// TwinCAT 3 PLC project Test
// ProgramVersion: 3.1.4020.10
// libraries:
//   Tc2_MC2, * (Beckhoff Automation GmbH)
//   Tc2_SerialCom, * (Beckhoff Automation GmbH)
//   Tc2_Standard, * (Beckhoff Automation GmbH)
//   Tc2_System, * (Beckhoff Automation GmbH)
//   Tc2_TcpIp, * (Beckhoff Automation GmbH)
//   Tc2_Utilities, * (Beckhoff Automation GmbH)
//   Tc3_Module, * (Beckhoff Automation GmbH)
// project tree:
//   DUTs/ ASCII.TcDUT, Boat.TcDUT
//   GVLs/ GVL_Const.TcGVL, IO.TcGVL
//   / PlcTask.TcTTO
//   POUs/ MAIN.TcPOU
//   POUs/model/ FB_AXIS.TcPOU, FB_Object.TcPOU, FB_RobotCom.TcPOU, FB_String.TcPOU, F_Messages.TcPOU, FB_TP.TcPOU, PRG_Com.TcPOU

CONFIGURATION Test
    RESOURCE PLC ON TwinCAT3
        TASK PlcTask(INTERVAL := T#10ms, PRIORITY := 20);
        PROGRAM MAIN WITH PlcTask : MAIN;
    END_RESOURCE
END_CONFIGURATION

// ---- DUTs/ASCII.TcDUT
TYPE ASCII :
STRUCT	
	AscByte			:ARRAY[1..5] OF BYTE;
END_STRUCT
END_TYPE

// ---- DUTs/Boat.TcDUT
//{attribute 'pack_mode' :='1'}
TYPE Boat :
STRUCT
	ID				: LREAL;			//ID
	CoolTime		: LREAL ;			//冷却时间
	BoatErrHandle	: LREAL ;			//报警舟处理：0未确认1回炉工艺2到自动化检查
	UseTimes		: LREAL ;			//使用次数
	bWaferLoad		: BOOL ;			//装片
	bJobDone		: BOOL ;			//工艺完成
	bCool			: BOOL ;			//冷却完成
	bNeedWash		: BOOL ;			//清洗		
	bError			: BOOL ;			//报警
	bReserve		: BOOL ;			//新舟 	
END_STRUCT
END_TYPE

// ---- GVLs/GVL_Const.TcGVL
{attribute 'qualified_only'}
VAR_GLOBAL
	
END_VAR

// ---- GVLs/IO.TcGVL
{attribute 'qualified_only'}
VAR_GLOBAL
	//Axisx_io: Tc2_MC2.AXIS_REF;
	IoTest 		AT %IB100 		: ARRAY[1..20] OF UINT;
	IoTest1		AT %QB100 	: ARRAY[1..20] OF UINT;
END_VAR

// ---- POUs/MAIN.TcPOU
PROGRAM MAIN
VAR
	AxisX				:FB_AXIS;
	Jogtest				:BOOL;
	bJOGPlus			:BOOL;
	bpower				:BOOL;
	ss,ss1				:STRING;
	var1,var2,var3		:INT;
	rvar1				:LREAL;
	iloop				:INT;
	rlayer				:REAL;
	bpttest				:BOOL;
	pttest1				:FB_TP;
	ptTest				:TP;
	ptout				:BOOL;
	ptin				:BOOL;
	rpttest				:R_TRIG;
	ttest				:TIME;
	bGetNetId			:BOOL:=FALSE;
	NullId				: T_AmsNetID:='0.0.0.0.0.0';
	bEnableCerDis		: BOOL;
	NT_StartProcess		: NT_StartProcess;
	NetId: T_AmsNetID;
	GetLocalAmsNetId: FB_GetLocalAmsNetId;	
	CPJ_DataTrans		:FB_RobotCom;
	PlcTaskSysInfo		: PlcTaskSystemInfo ;			//系统任务信息	
	ss11:STRING(6);
	ss12:STRING(1);
	Out_BoatID:BYTE;
	W:WORD;
	mystr:FB_String;
	i:UINT;
	StrToSend:STRING;
	I1:INT;
END_VAR

//W:=10;
//ss:=WORD_TO_HEXSTR(in:= W, iPrecision:= 2, bLoCase:= FALSE);
//M_PT();
//Init();
//M_Axis();
//CPJ_DataTrans.M_Run();
//mystr.A_Run();
//StrToSend:= CONCAT(CONCAT(CONCAT(CONCAT('@0',INT_TO_STRING(I1)),
//							Chr(16#2)), 'RFV'), Chr(16#3));
//Out_BoatID:=Tc2_SerialCom.ASC(str:=ss11);
//mid(ss11,1,1);
FOR iloop:=1 TO 5 DO
	iloop:=iloop-1;
END_FOR
I1:=ss[iloop];
iloop:=1;

ACTION Init:
IF NOT bGetNetId THEN
	GetLocalAmsNetId(bExecute:= TRUE, tTimeOut:= T#300MS, AddrString=> NetId);	
	IF GetLocalAmsNetId.bBusy OR GetLocalAmsNetId.bError OR NetId=NullId THEN
		GetLocalAmsNetId(bExecute:= FALSE);
	END_IF
	IF NOT(NetId= NullId)THEN
		NT_StartProcess(NETID:= NetId, PATHSTR:='\windows\CerDisp.exe' , 
					DIRNAME:= '\windows', 	START:= TRUE);
		bGetNetId:=TRUE;
	END_IF
END_IF
END_ACTION

METHOD M_Axis : BOOL
VAR_INPUT
	bStartTest:BOOL;
	
END_VAR
VAR
	iStep:INT;
	
END_VAR

AxisX.AxisId:='AxisX';
AxisX.bPowerCmd:=TRUE;

AxisX.JogAcc:=10;
AxisX.JogDec:=10;
AxisX.JogVel:=1;
AxisX.JogDis:=100;
AxisX.rHomeBackDis:=-5;
AxisX.rHomeOffset:=20;
AxisX.M_Run();


CASE iStep OF
	0:
		;
	1:
	;
	2:
	;

END_CASE
END_METHOD

 METHOD M_PT : BOOL
VAR_INPUT
END_VAR

ptTest(IN:= ptin, PT:=T#60S , Q=> ptout, ET=> );

pttest1(Pt:=T#60S , In:=bpttest );
rpttest(CLK:=pttest1.Out , Q=> );
IF rpttest.Q THEN
	var1:=var1+1;
END_IF
IF pttest1.Q THEN
	var2:=var2+1;
END_IF
END_METHOD

END_PROGRAM

// ---- POUs/model/FB_AXIS.TcPOU
FUNCTION_BLOCK FB_AXIS
VAR_INPUT
	
	AxisId			:STRING(10);
	iMode			:INT;
//CMD
	bMoveOk			:BOOL;
	bPowerCmd		:BOOL;
	bResetCmd		:BOOL;
	bJogPCmd		:BOOL;
	bJogNCmd		:BOOL;
	bMovPosCmd		:BOOL;	
	bStopCmd		:BOOL;
	bHomeCmd		:BOOL;	
	bMoveVelPCmd	:BOOL;
	bMoveVelNCmd	:BOOL;	
//para          	
	JogVel			:LREAL;
	JogDis			:LREAL;
	JogAcc			:LREAL;
	JogDec			:LREAL;
	MovVel			:LREAL;
	TargetPos		:LREAL;
	MovAcc			:LREAL;
	MovDec			:LREAL;
//pospara
	rForewardPos	:REAL;	
	rHomeVel1		:INT:=10;
	rHomeVel2		:INT:=5;
	rHomeBackDis	:INT;	
	rHomeOffset		:INT;
//signal
	bHomeSignal		:BOOL;		//原点位
	bForewardSignal	:BOOL;		//进到位
	bBackwardSignal	:BOOL;		//退到位
	bBackLimit		:BOOL;		//后限位
	bForeLimit		:BOOL;		//前限位
END_VAR
VAR_OUTPUT
	bHomed			:BOOL;		//轴初始化完成
	bEnable			:BOOL;		//轴使能成功
	bMoving			:BOOL;		//轴运动中
	bBusy			:BOOL;		//busy时不能接收新的运动指令，只能先stop
	ActPos			:LREAL;		//编码器位置
	ActSpeed		:LREAL;
	ActTorque		:LREAL;
	
	bPowerDone		:BOOL;		
	bPowerError		:BOOL;	
	bJogDone		:BOOL;
	bJogError		:BOOL;	
	bMovDone		:BOOL;
	bMovError		:BOOL;	
	bResetDone		:BOOL;
	bResetError		:BOOL;
	bStopDone		:BOOL;
	bStopError		:BOOL;
	bVelReached		:BOOL;
	bMoveVelError	:BOOL;
	
	bErr			:ARRAY[1..20] OF BOOL;
	//1:负极限不能反向点动			2：正极限不能正向点动
	//3：轴未初始化，不能运动		4：不满足运动条件，有碰撞风险
	//5：编码器位置和开关不一致		6：轴使能消失
	//7：轴扭矩超过设置值			8:到极限不能运动
	//:
	
	bAtHomePos		:BOOL;
	bAtForeWardPos	:BOOL;
	
END_VAR
VAR
	Axis			: axis_ref;
	Power			: Tc2_MC2.MC_Power ;
	JOGH			: Tc2_MC2.MC_MoveRelative;
	JOG				: Tc2_MC2.MC_MoveRelative;
	MoveA			: Tc2_MC2.MC_MoveAbsolute;
	MoveVH			: Tc2_MC2.MC_MoveVelocity;	//Homing movv
	MoveV			: Tc2_MC2.MC_MoveVelocity;
	Reset			: Tc2_MC2.MC_Reset;
	Stop			: Tc2_MC2.MC_Stop;
	StopLimit		: Tc2_MC2.MC_Stop;
	SetPos			: Tc2_MC2.MC_SetPosition;	
	WritePara		: MC_WriteParameter;
	Update			: MC_ReadStatus ;
	tErr			: ARRAY[1..20] OF TON;
	
//home
	rHome			: Tc2_Standard.R_TRIG;
	Home_Done		:BOOL;
	Home_Error		:BOOL;
	HomeState		:INT;
	Home_bError		:ARRAY[0..10] OF BOOL;
	Home_bDone		:ARRAY[0..10] OF BOOL;
	tHomeStep		:ARRAY[0..10] OF Ton;
END_VAR

METHOD M_Home : BOOL
VAR
	iLoop		:INT;
END_VAR
//初始化过程的变量初始化
	rHome(CLK:=bHomeCmd  , Q=> );
	IF rHome.Q THEN
		bHomed :=FALSE;
		Home_Done:=FALSE;
		Home_Error:=FALSE;
		HomeState:=0;		
		FOR iLoop:=0 TO 10 DO
			Home_bError[iLoop]:=FALSE;
			Home_bDone[iLoop]:=FALSE;
		END_FOR
		SetPos(	Axis:=Axis ,Execute:=FALSE);
		MoveVH(Axis:= Axis ,Execute:= FALSE);
		STOP(Axis :=Axis ,Execute :=FALSE );
		JOGH(Axis :=Axis ,Execute :=FALSE );
	END_IF

//初始化过程
	IF bHomeCmd THEN		
		CASE HomeState OF
			0:			
				HomeState:=1;								
			1:
				IF NOT bHomeSignal THEN					
					MoveVH(Axis:=Axis ,Execute:= TRUE, Velocity:=rHomeVel1 ,Acceleration:=rHomeVel1*5,
					Direction:=MC_Negative_Direction , Error=> Home_bError[0] );
				ELSE
					MoveVH(Axis:= Axis ,Execute:= FALSE);					
					STOP(Axis :=Axis ,Execute :=TRUE, Deceleration:=rHomeVel1*10,Done=>Home_bDone[1]);
					IF Home_bDone[1] THEN
						STOP(Axis :=Axis ,Execute :=FALSE);												
						HomeState:=2;												
					END_IF					
				END_IF
			2:				
				IF bHomeSignal THEN				
					MoveVH(Axis:=Axis ,Execute:= TRUE, Velocity:=rHomeVel2 ,Direction:=MC_Positive_Direction);									
				ELSE
					MoveVH(Axis:=Axis ,Execute:= FALSE);	
					STOP(Axis :=Axis ,Execute :=TRUE,Deceleration:=rHomeVel2*15, Done=>Home_bDone[2]);						
					IF Home_bDone[2] THEN						
						STOP(Axis :=Axis ,Execute :=FALSE);											
						HomeState:=3;																							
					END_IF						
				END_IF
			3:					
				JOGH(Axis:=Axis, Execute:= TRUE, Distance:=rHomeBackDis,Velocity:=1 , Done=> Home_bDone[3]);
				IF Home_bDone[3] THEN
					Home_bDone[4]:=TRUE;
				END_IF
				IF Home_bDone[4] THEN					
					JOGH(Axis:=Axis ,Execute:= FALSE);	
					STOP(Axis :=Axis ,Execute :=TRUE,Deceleration:=20, Done=>Home_bDone[5]);
					IF Home_bDone[5] THEN
						HomeState:=4;
					END_IF					
				END_IF	
			4:
				SetPos(	Axis:=Axis,Execute:= TRUE,Position:=80,Mode:=FALSE , Done=>Home_bDone[6]);				
				IF Home_bDone[6] THEN
					SetPos(Axis:=Axis,Execute:= FALSE);
					HomeState:=0;												
					bHomed :=TRUE;
					bHomeCmd := FALSE;							
					bResetCmd :=TRUE ;
				END_IF				
		END_CASE		
	END_IF
END_METHOD

METHOD M_Home1 : BOOL
VAR
	iLoop	:INT;
END_VAR
//初始化过程的变量初始化
	rHome(CLK:=bHomeCmd  , Q=> );
	IF rHome.Q THEN
		bHomed :=FALSE;
		Home_Done:=FALSE;
		Home_Error:=FALSE;
		HomeState:=0;		
		FOR iLoop:=0 TO 10 DO
			Home_bError[iLoop]:=FALSE;
			Home_bDone[iLoop]:=FALSE;
			tHomeStep[iLoop](IN:=FALSE , PT:= , Q=> , ET=> );
		END_FOR
		SetPos(	Axis:=Axis ,Execute:=FALSE);
		MoveVH(Axis:= Axis ,Execute:= FALSE);
		STOP(Axis :=Axis ,Execute :=FALSE );
		JOGH(Axis :=Axis ,Execute :=FALSE );
	END_IF

//初始化过程
	IF bHomeCmd THEN		
		CASE HomeState OF
			0:			
				HomeState:=1;								
			1:
				IF NOT bHomeSignal AND NOT bBackwardSignal THEN					
					MoveVH(Axis:=Axis ,Execute:= TRUE, Velocity:=rHomeVel1 ,Acceleration:=rHomeVel1*5,
					Direction:=MC_Negative_Direction , Error=> Home_bError[0] );
				ELSE
					MoveVH(Axis:= Axis ,Execute:= FALSE);					
					STOP(Axis :=Axis ,Execute :=TRUE, Deceleration:=rHomeVel1*20,Done=>Home_bDone[1]);
					IF Home_bDone[1] THEN
						STOP(Axis :=Axis ,Execute :=FALSE);	
						IF bHomeSignal THEN										
							HomeState:=3;	
						ELSIF bBackwardSignal THEN
							HomeState:=2;
							Home_bDone[1]:=FALSE;
						END_IF 										
					END_IF					
				END_IF
			2:
				JOGH(Axis:=Axis, Execute:= TRUE, Distance:=rHomeOffset+10,Velocity:=rHomeVel1 , Done=> Home_bDone[2]);
				IF Home_bDone[2] THEN
					Home_bDone[3]:=TRUE;
				END_IF
				IF Home_bDone[3] THEN					
					JOGH(Axis:=Axis ,Execute:= FALSE);	
					//STOP(Axis :=Axis ,Execute :=TRUE,Deceleration:=20, Done=>Home_bDone[4]);
					Home_bDone[4]:=TRUE;
					IF Home_bDone[4] THEN
						HomeState:=1;
						STOP(Axis :=Axis ,Execute :=FALSE);	
					END_IF					
				END_IF					
			3:				
				IF bHomeSignal THEN				
					MoveVH(Axis:=Axis ,Execute:= TRUE, Velocity:=rHomeVel2 ,Direction:=MC_Positive_Direction);									
				ELSE
					MoveVH(Axis:=Axis ,Execute:= FALSE);	
					STOP(Axis :=Axis ,Execute :=TRUE,Deceleration:=rHomeVel2*25, Done=>Home_bDone[5]);						
					IF Home_bDone[5] THEN						
						STOP(Axis :=Axis ,Execute :=FALSE);							
						HomeState:=4;																																		
					END_IF						
				END_IF
			4:					
				JOGH(Axis:=Axis, Execute:= TRUE, Distance:=rHomeBackDis,Velocity:=1 , Done=>Home_bDone[6]);
				IF Home_bDone[6] THEN
					Home_bDone[7]:=TRUE;
				END_IF
				IF Home_bDone[7] THEN					
					JOGH(Axis:=Axis ,Execute:= FALSE);	
					//STOP(Axis :=Axis ,Execute :=TRUE,Deceleration:=20, Done=>Home_bDone[8]);
					
					//IF Home_bDone[8] THEN
					HomeState:=5;
					//END_IF					
				END_IF	
			5:
				SetPos(	Axis:=Axis,Execute:= TRUE,Position:=rHomeOffset,Mode:=FALSE , Done=>Home_bDone[9]);				
				IF Home_bDone[9] THEN
					SetPos(Axis:=Axis,Execute:= FALSE);
					HomeState:=0;												
					bHomed :=TRUE;
					bHomeCmd := FALSE;							
					bResetCmd :=TRUE ;
				END_IF				
		END_CASE		
	END_IF
END_METHOD

METHOD M_Init : BOOL
VAR_INPUT
END_VAR
END_METHOD

METHOD M_MovDis : BOOL
VAR_INPUT
END_VAR
IF bJogPCmd THEN
	JOG(Axis:=Axis ,Execute:= TRUE,	Distance:=JogDis , 
	Velocity:=JogVel , Acceleration:=JogAcc ,Deceleration:=JogDec , 	
	Done=> bJogDone, Error=>bJogError );
	IF bJogDone OR bJogError THEN
		bJogPCmd:=FALSE;		
		JOG(Axis:=Axis ,Execute:= FALSE);
	END_IF
	IF bForeLimit THEN
		bErr[2]:=TRUE;
		bJogNCmd:=FALSE;
		StopLimit(Axis:=Axis ,Execute:=TRUE,Deceleration:=JogVel*20);		
		JOG(Axis:=Axis ,Execute:= FALSE);
	END_IF
ELSIF bJogNCmd THEN
	JOG(Axis:=Axis ,Execute:= TRUE,	Distance:=0-JogDis , 
	Velocity:=JogVel , Acceleration:=JogAcc ,Deceleration:=JogDec , 	
	Done=> bJogDone, Error=>bJogError );
	IF bJogDone OR bJogError THEN
		bJogNCmd:=FALSE;		
		JOG(Axis:=Axis ,Execute:= FALSE);
	END_IF	
	IF bBackLimit THEN
		bErr[1]:=TRUE;
		bJogPCmd:=FALSE;
		StopLimit(Axis:=Axis ,Execute:=TRUE,Deceleration:=JogVel*20);		
		JOG(Axis:=Axis ,Execute:= FALSE);
	END_IF
ELSE
	JOG(Axis:=Axis ,Execute:= FALSE);
END_IF
IF bBackLimit OR bForeLimit THEN
	StopLimit(Axis:=Axis ,Execute:=FALSE);	
END_IF
END_METHOD

METHOD M_MoveVel : BOOL
VAR_INPUT
END_VAR
IF bMoveVelPCmd THEN
	MoveV(Axis:=Axis ,Execute:= TRUE, Velocity:= MovVel, 
	Acceleration:=MovAcc , 	Deceleration:=MovDec , 	Direction:= Tc2_MC2.MC_Positive_Direction,	 
	InVelocity=>bVelReached, 	Busy=> , 	Active=> , 	CommandAborted=> , 	Error=>bMoveVelError, 	ErrorID=> );
	IF bMoveVelError THEN
		MoveV(Axis:=Axis ,Execute:= FALSE);
	END_IF
	bMoveVelPCmd:=FALSE;
ELSIF bMoveVelNCmd THEN
	MoveV(Axis:=Axis ,Execute:= TRUE, Velocity:= MovVel, 
	Acceleration:=MovAcc , 	Deceleration:=MovDec , 	Direction:= Tc2_MC2.MC_Positive_Direction,	 
	InVelocity=>bVelReached, 	Busy=> , 	Active=> , 	CommandAborted=> , 	Error=>bMoveVelError, 	ErrorID=> );
	IF bMoveVelError THEN
		MoveV(Axis:=Axis ,Execute:= FALSE);
	END_IF
ELSE
	MoveV(Axis:=Axis ,Execute:= FALSE);
END_IF
END_METHOD

METHOD M_MovPos : BOOL
VAR_INPUT
END_VAR
IF bMovPosCmd THEN
	MoveA(Axis:=Axis ,Execute:=TRUE , Position:=TargetPos , 
	Velocity:=MovVel, Acceleration:=MovAcc , Deceleration:=MovDec ,	
	Done=>bMovDone ,Error=>bMovError);
	IF bMovDone OR bMovError THEN
		//MoveA(Axis:=Axis ,Execute:=FALSE);
		//bMovCmd:=FALSE;
	END_IF
ELSE
	MoveA(Axis:=Axis ,Execute:=FALSE);
END_IF
END_METHOD

METHOD M_Power : BOOL
VAR_INPUT
END_VAR
Power(	Axis:=Axis ,
		Enable:=bPowerCmd , 
		Enable_Positive:=TRUE ,
		Enable_Negative:=TRUE ,
		Override:=100 ,
		Error=>bPowerError);
END_METHOD

METHOD M_Process : BOOL
VAR_INPUT
END_VAR
END_METHOD

METHOD M_Reset : BOOL
VAR_INPUT
END_VAR
IF bResetCmd THEN
	Reset(Axis:= Axis, Execute:= TRUE, 
	Done=>bResetDone ,Error=> bResetError );
	IF bResetDone OR bResetError THEN
		bResetCmd:=FALSE;
		Reset(Axis:= Axis, Execute:=FALSE);
	END_IF
	
	bPowerError	:=FALSE;	
	bJogError	:=FALSE;	
	bMovError	:=FALSE;	
	bResetError	:=FALSE;
	bStopError	:=FALSE;
ELSE
	Reset(Axis:= Axis, Execute:=FALSE);
END_IF
END_METHOD

METHOD M_Run : BOOL
VAR_INPUT
END_VAR
M_Update();
M_Power();
M_Reset();
M_Stop();
M_MovPos();
M_MovDis();
M_MoveVel();
M_Home1();
END_METHOD

METHOD M_Stop : BOOL
VAR_INPUT
END_VAR
IF bStopCmd THEN
	bJogPCmd:=FALSE;
	bJogNCmd:=FALSE;
	bMovPosCmd	:=FALSE;
	bHomeCmd:=FALSE;
	Stop(Axis:= Axis, Execute:= TRUE, Deceleration:= MovDec*10, 
	Done=>bStopDone ,Error=> bStopError );
	
	IF bStopDone OR bStopError THEN
		bStopCmd:=FALSE;
		Stop(Axis:= Axis, Execute:=FALSE);
	END_IF
ELSE
	Stop(Axis:= Axis, Execute:=FALSE);
END_IF
END_METHOD

METHOD M_Update : BOOL
VAR
	iLoop		:INT;	
END_VAR
//到达极限则复位点动指令，并报错
IF bBackLimit AND bJogNCmd THEN	
	bErr[1]:=TRUE;
	{text'负极限不能负向点动'}
END_IF
IF bforeLimit AND bJogPCmd THEN	
	bErr[2]:=TRUE;
	{text'正极限不能正向点动'}
END_IF
//点动错误自动复位
FOR iLoop:=1 TO 2 DO
	tErr[iLoop](IN:=bErr[iLoop] , PT:=T#10S);
	IF tErr[iLoop].Q THEN
		bErr[iLoop]:=FALSE;
	END_IF
END_FOR

//到极限不能运动
IF bBackLimit OR bforeLimit THEN
	IF bMovPosCmd THEN
		bMovPosCmd:=FALSE;
		bErr[8]:=TRUE;
	END_IF	
END_IF

//未初始化不能运动
IF NOT bHomed THEN
	IF bMovPosCmd THEN
		bMovPosCmd:=FALSE;
		bErr[3]:=TRUE;
	END_IF
END_IF

//状态更新
Update(Axis:=Axis ,Enable:=TRUE);
ActPos:=Axis.NcToPlc.ActPos;
ActSpeed:=Axis.NcToPlc.ActVelo;
ActTorque:=Axis.NcToPlc.ActTorque;
bEnable:=Axis.NcToPlc.StateDWord.20;
bBusy:=bJogNCmd OR bJogPCmd OR bMovPosCmd OR bMoveVelPCmd OR bMoveVelNCmd OR bHomeCmd;
bMoving:=Update.Status.Moving;
END_METHOD

END_FUNCTION_BLOCK

// ---- POUs/model/FB_TP.TcPOU
FUNCTION_BLOCK FB_TP
VAR_INPUT
	Pt:TIME;
	In:BOOL;
END_VAR
VAR_OUTPUT
	Out:BOOL;
	Q	:BOOL;
END_VAR
VAR
	bfyk	:BOOL;
	T1,T2	:TON;
	rOut	:R_TRIG;	
END_VAR

IF In THEN
	T1(IN:=NOT bfyk , PT:= Pt, Q=> , ET=> );
	IF T1.Q THEN
		bfyk:=TRUE;
	END_IF
	T2(IN:=bfyk , PT:= Pt, Q=> , ET=> );
	IF T2.Q THEN
		bfyk:=FALSE;
	END_IF
	Out :=bfyk;
	rOut(CLK:=Out , Q=>Q );
ELSE
	Out :=FALSE;
END_IF

END_FUNCTION_BLOCK

// ---- POUs/model/FB_RobotCom.TcPOU
FUNCTION_BLOCK FB_RobotCom
(*
	插片机通讯 模块
	1.作为服务器
	2.客户端——二所
	3.客户端-江松
*)
VAR_INPUT
	bReconnectCmd		:BOOL;	
	PEData				:ARRAY[1..30] OF UINT;		//写入的PE数据
	iServer				:INT;	
END_VAR
VAR_OUTPUT
	bError				:ARRAY[1..10] OF BOOL;		//1:连接错误，2读写错误或者超时
	RobotData			:ARRAY[1..30] OF UINT;		//读出的JS数据
	bConnected			:BOOL;						//通讯正常
END_VAR
VAR
	DataNull			:ARRAY[1..30] OF UINT;		//0
//1.AS Server	


//AS Client
//公用	
	tcpconnect			:FB_SocketConnect;			//
    tcpclose			:FB_SocketClose;			//
    tcpcloseall			:FB_SocketCloseAll;			//
	tcpsend				:FB_SocketSend;				//
    tcpreceive			:FB_SocketReceive;			//
	hSocket				:T_HSOCKET;
	
	close_do			:BOOL;						//
	closeall_do			:BOOL;   					//
	connect_do			:BOOL:=TRUE;	
	Connect_error		:BOOL;	
	bsenderror			:BOOL;
	breceiveerror		:BOOL;
	bsendbusy			:BOOL;
	brecvbusy			:BOOL;
	
	tReadWriteErr		:TON;
	bReadWriteErr		:BOOL;
	tReadWriteOK		:TON;
	bReadWriteOK		:BOOL;
	
	tConnected			:TON;
	tCon_ErrorConfirm	:TON;
	tConnect_error		:TON;
	tConnect_error1		:TON;
	rReconnect			:R_TRIG;	
	ServerIp			:STRING;
	iPort				:UDINT;

	iReconStep			:INT;
	tRecon				:ARRAY[0..2] OF TON;

	

	
//robo-tec 
	iRunStepRT			:INT;
		
	arrSendDataRT		:ARRAY[1..30] OF BYTE;
	arrRecieveDataRT	:ARRAY[1..30] OF BYTE;
	tStepRT				:ARRAY[0..1] OF TON;	
	iSendTimes			:INT;	

	//robo-tec 11
	iRunStepRT1			:INT;
		
	arrSendDataRT1		:STRING(20);
	arrRecieveDataRT1	:STRING(20);
	tStepRT1			:ARRAY[0..1] OF TON;	
	iSendTimes1			:INT;	
//JS ADS

END_VAR

METHOD M_Connect : BOOL
VAR
END_VAR
//connnect
	tcpconnect(sSrvNetId:='' ,	sRemoteHost:=ServerIp ,nRemotePort:=iPort,
		bExecute:=connect_do ,	tTimeout:=T#5S ,bError=>Connect_error );
	//连续10s无连接错误认为连接成功	
	tConnected(IN:= NOT Connect_error, PT:=T#10S , Q=>bConnected , ET=> );
	bError[1]:=NOT bConnected;
//recoonect	读写错误或连接错误时，自动重连
	IF NOT bReconnectCmd THEN
		tConnect_error(IN:= Connect_error OR NOT bReadWriteOK,PT:=T#60S);
	END_IF	
	rReconnect(CLK:=tConnect_error.Q , Q=> );	
	IF rReconnect.Q THEN
		bReconnectCmd:=TRUE;
	END_IF
	
	IF bReconnectCmd THEN
		CASE iReconStep OF
			0:
				connect_do:=FALSE;
				tcpCloseAll(sSrvNetId:= ,bExecute:=TRUE );			
				tRecon[0](IN:=TRUE , PT:=T#1S , Q=> , ET=> );				
				IF tRecon[0].Q THEN
					iReconStep:=1;
					tRecon[0](IN:=FALSE);
					tcpCloseAll(sSrvNetId:= ,bExecute:=FALSE );
				END_IF
			1:
				connect_do:=TRUE;							
				tRecon[1](IN:=TRUE , PT:=T#1S , Q=> , ET=> );	
				IF tRecon[1].Q THEN
					iReconStep:=0;
					tRecon[1](IN:=FALSE);
					tConnect_error(IN:= FALSE);
					bReconnectCmd:=FALSE;
				END_IF
		END_CASE
	END_IF
END_METHOD

METHOD M_DataMake : BOOL
VAR
	iloop:INT;
END_VAR
arrSendDataRT1:='';
FOR iloop:=1 TO 30 DO
	//arrSendDataRT1:=arrSendDataRT1+BOOL_TO_STRING(UINT_TO_BOOL(PEData[iloop]));
	//arrSendDataRT1:=CONCAT(arrSendDataRT1,UINT_TO_STRING(PEData[iloop]));
	arrSendDataRT[iloop]:=UINT_TO_BYTE(PEData[iloop]);
END_FOR
END_METHOD

METHOD M_RT1_DataTrans : BOOL
VAR
	iLoop:INT;
END_VAR
//循环读写过程	
	CASE iRunStepRT1 OF 	
		0://发送数据
			M_DataMake();	
				
			IF 	iSendTimes=0 THEN	
				tcpSend(sSrvNetId:='' ,
						hSocket:=tcpconnect.hSocket,
						cbLen:= SIZEOF(arrSendDataRT),
						pSrc:=ADR(arrSendDataRT),
						bExecute:= TRUE,
						tTimeout:=T#5S,
						bError=>bsenderror,
						bBusy=>bsendbusy);
			END_IF
			tStepRT1[0](IN:=TRUE,PT:=T#120MS);
			IF tStepRT1[0].Q THEN							
				iRunStepRT1:=1;
				tcpSend(hSocket:=tcpconnect.hSocket,bExecute:=FALSE);
				tStepRT1[0](IN:=FALSE );
				iSendTimes1:=iSendTimes1+1;
				IF iSendTimes1=6 THEN
					iSendTimes1:=0;
				END_IF
			END_IF				
		1://接收数据					
			tcpReceive(sSrvNetId:='',
					   hSocket:=tcpconnect.hSocket,
					   cbLen:=SIZEOF(arrRecieveDataRT),
					   pDest:=ADR(arrRecieveDataRT),
					   bExecute:=TRUE,
					   tTimeout:=T#5S,
					   bError=>breceiveerror,
					   bBusy=>brecvbusy);
			tStepRT1[1](IN:=TRUE,PT:= T#120MS);
			IF tStepRT1[1].Q THEN											
				tStepRT[1](IN:=FALSE );
				tcpreceive(hSocket:=tcpconnect.hSocket,bExecute:=FALSE);
				iRunStepRT1:=0;
			END_IF		
	END_CASE

	tReadWriteErr(IN:=bsenderror OR bsendbusy OR breceiveerror OR brecvbusy OR bError[2],
				  PT:=T#0.5S , Q=>bReadWriteErr);
	tReadWriteOK(IN:=NOT bReadWriteErr , PT:=T#10S , Q=>bReadWriteOK , ET=> );
END_METHOD

METHOD M_Run : BOOL
IF iServer=0 THEN		
		iPort:=8501;
		ServerIp:='192.168.1.12';
		M_Connect();
		IF NOT Connect_error THEN	
			M_RT1_DataTrans();
			IF bReadWriteErr THEN
				RobotData:=DataNull;
			END_IF		
		ELSE
			RobotData:=DataNull;	
		END_IF
	END_IF
END_METHOD

END_FUNCTION_BLOCK

// ---- POUs/model/FB_String.TcPOU
FUNCTION_BLOCK FB_String
VAR_INPUT
	S_BoatID	:STRING(6);
	PE_BoatID:UINT;	
	RB_BoatID 	:ARRAY[0..6] OF BYTE;
	TubeIP		:ARRAY[1..5] OF INT;
END_VAR
VAR_OUTPUT
	rbboatid:INT;
	Tubenetid	:ARRAY[1..5] OF STRING;
	B_BoatID	:ARRAY[0..6] OF BYTE;
	 
END_VAR
VAR
	istrLen,iLoop:INT;
	strout:STRING;
	PE_BoatIDRB:ARRAY[0..6] OF BYTE;
	strBoatId:STRING;
	str:STRING;
	arrstrId	:ARRAY[1..6] OF STRING;
	
	
END_VAR

ACTION A_Run:
//str2byte
	strBoatId:=UINT_TO_STRING(PE_BoatID);
	istrLen:=LEN(strBoatId);
	FOR iLoop:=0 TO 6 DO
		PE_BoatIDRB[iLoop]:=0;
	END_FOR
	FOR iLoop:=0 TO istrLen DO
		PE_BoatIDRB[iLoop]:=strBoatId[iLoop];
	END_FOR

//byte2str
	strout:='';
	FOR iLoop:=1 TO 6 DO
		arrstrId[iLoop]:=BYTE_TO_STRING(PE_BoatIDRB[iLoop]);
		strout:=CONCAT(strout,arrstrId[iLoop]);			
	END_FOR
	rbboatid:=STRING_TO_INT(strout);
	
	
	
//tubenetid
	FOR iLoop:=1 TO 5 DO
		Tubenetid[iloop]:=CONCAT(INT_TO_STRING(TubeIP[1]),'.');
		Tubenetid[iloop]:=CONCAT(Tubenetid[iloop],CONCAT(INT_TO_STRING(TubeIP[2]),'.'));
		Tubenetid[iloop]:=CONCAT(Tubenetid[iloop],CONCAT(INT_TO_STRING(TubeIP[3]),'.'));
		Tubenetid[iloop]:=CONCAT(Tubenetid[iloop],CONCAT(INT_TO_STRING(TubeIP[4]+iloop-1),'.1.1'));
	END_FOR
END_ACTION

END_FUNCTION_BLOCK

// ---- POUs/model/FB_Object.TcPOU
FUNCTION_BLOCK FB_Object
VAR_INPUT
END_VAR
VAR_OUTPUT
END_VAR
VAR
	iMem:UINT;
END_VAR

METHOD PUBLIC M_Add : UINT
VAR_INPUT
	iVal:UINT;
END_VAR
iMem:=iMem+iVal;
M_Add:=iMem;
END_METHOD

PROPERTY PUBLIC P_Memory : uint
GET
P_Memory:=iMem;
END_GET
SET
iMem:=P_Memory;
END_SET
END_PROPERTY

END_FUNCTION_BLOCK

// ---- POUs/model/F_Messages.TcPOU
FUNCTION F_Messages : BOOL
VAR_INPUT
END_VAR
VAR
END_VAR

;
{text'hello world'}
{info'information'}
{warn'warning'}
//{error'Error!'}

END_FUNCTION

// ---- POUs/model/PRG_Com.TcPOU
PROGRAM PRG_Com
VAR
	i :INT;
END_VAR

METHOD M_Add : BOOL
VAR_INPUT
END_VAR
i:=i+1;
END_METHOD

END_PROGRAM
